// TIA Portal V17 export
// export: Created 2024-08-09T12:53:19.0565445Z, ExportSetting WithDefaults, DisplayName Totally Integrated Automation Portal, DisplayVersion V17 Update 7, DisplayName TIA Portal Openness, DisplayVersion V17 Update 7, DisplayName TIA Portal Version Control Interface, DisplayVersion V17, DisplayName STEP 7 Professional, DisplayVersion V17 Update 7, DisplayName STEP 7 Safety, DisplayVersion V17 Update 6, DisplayName WinCC Professional, DisplayVersion V17 Update 7
TYPE "S_Exp_Dos"
// stored: IsFailsafeCompliant false
   STRUCT
      Pt_Zs : "S_Suivi_Dosage";
      CommunDos : "S_Dosage_Commun";
      Pt_Cel : USInt;
      ChNoeud : "S_ChngNoeud";
      Cir : "S_Circuit";
      Cir_Sans_Test_Reserve : "S_Circuit";
      Nouv_Circuit : "S_Circuit";
      Dial_Def : "S_DIALOG_DEF";
      Lst_Taches_Amont_Qte : Array[0.."T_MAX_AMONTAVAL"] of SInt;
      Lst_Taches_Aut_Dem { ExternalAccessible := 'False'; ExternalVisible := 'False'; ExternalWritable := 'False'} : Array[0.."T_MAX_AMONTAVAL"] of "S_TacheNiv";
      Lst_Taches_Att_Fin_Amont { ExternalAccessible := 'False'; ExternalVisible := 'False'; ExternalWritable := 'False'} : Array[0.."T_MAX_AMONTAVAL"] of "S_TacheNiv";
      Lst_Taches_Arret_Test_NH { ExternalAccessible := 'False'; ExternalVisible := 'False'; ExternalWritable := 'False'} : Array[0.."T_MAX_AMONTAVAL"] of "S_TacheNiv";
      _DestEc : "S_Cellule";
      CntlDest { ExternalAccessible := 'False'; ExternalVisible := 'False'; ExternalWritable := 'False'} : Struct
         Etape { ExternalAccessible := 'False'; ExternalVisible := 'False'; ExternalWritable := 'False'} : SInt;
         EtapeMemo { ExternalAccessible := 'False'; ExternalVisible := 'False'; ExternalWritable := 'False'} : SInt;
         EtpPrec { ExternalAccessible := 'False'; ExternalVisible := 'False'; ExternalWritable := 'False'} : SInt;
         TpsPicke { ExternalAccessible := 'False'; ExternalVisible := 'False'; ExternalWritable := 'False'} : Date_And_Time;
      END_STRUCT;
      Orig_Avec_Mls : String;
      Orig_Sans_Mls : String;
      Qte : Real;
      Debut_Exp : Date_And_Time;
      Debut_NH : Date_And_Time;
      Tps_Entre_Rech_Cir : Time;
      Tps_Avant_Relance_Cir : Time;
      Tps_Masque_NH : Time;
      Tps_Picke_NH : Date_And_Time;
      Tps_Att_Cir_Noeud : Time;
      _IndexDestEc : Int := -1;
      Mob_Suiv : Int := -1;
      Mob_Prec : Int := -1;
      Noeud : Int := -1;
      Orig : Int := -1;
      Num_Circuit : USInt;
      _TypeCelDest : USInt;
      _Cellule_Trouve : SInt;
      Tac_Amont : SInt := -1;
      Tac_Lanc_Exp : SInt := -1;
      Fg_Dest_Interm : Bool;
      Fg_Chg_Dest_Noeud : Bool;
      Fg_Aut_Chg_Cir : Bool;
      Fg_Arret_Amont : Bool;
      Fg_NH_Dest : Bool;
      Fg_Test_NH : Bool;
      Fg_Masq_NH : Bool;
      Fg_Ctrl_Incomp : Bool;
      Fg_Ctrl_Hopital : Bool;
      Fg_Ctrl_Stock : Bool;
      Fg_Intercep : Bool;
      Fg_Preposit : Bool;
      Fg_Cir_Enc : Bool;
      Fg_Chg_Dest_Enc : Bool;
      Fg_Melas : Bool;
      Fg_Chg_Dest_Serie_Dem : Bool;
      Fg_Lanc : Bool;
   END_STRUCT;
   // Lst_Taches_Amont_Qte[0..9] := -1;
END_TYPE
